FUNCTION Call_Remover

instFBRemover(PartPresent := RemoverPartPresent,
			  ActorInstanceIndex := 1,
			  ActorInstanceName := 'Remover conveyor',
			  HMIInterface := HMI.hmiMachineSectionInterface,
			  RemovePart => Remover);

END_FUNCTION

(* stored: Version 1.1.0.1
   POU Call_Remover: Id {124be3c7-c944-4f44-bd3e-c30afe3519a2}, SpecialFunc None *)
